// TIA Portal V20 export
// export: Created 2026-04-20T19:04:17.7701374Z, ExportSetting WithDefaults, DisplayName Totally Integrated Automation Portal, DisplayVersion V20, DisplayName TIA Portal Openness, DisplayVersion V20, DisplayName TIA Portal Version Control Interface, DisplayVersion V20, DisplayName STEP 7 Professional, DisplayVersion V20, DisplayName STEP 7 Safety, DisplayVersion V20, DisplayName WinCC Basic/Comfort/Advanced, DisplayVersion V20
TYPE "UDT_ProcessUnit"
// stored: IsFailsafeCompliant false
   STRUCT
      unitId : Int := 0;   // Unique unit identifier within the plant
      unitName : String[32] := 'Unit';   // Human-readable unit name
      recipeId : Int := 0;   // Active recipe identifier
      modules { S7_SetPoint := 'True'} : Array[1..3] of "UDT_EquipmentModule";   // Equipment modules within this unit
   END_STRUCT;
END_TYPE
